{attribute 'qualified_only'}
{attribute 'strict'}
TYPE Command_State :
(
	Exekute := 0,
	Wate := 1,
	Complete := 2,
	Error := 3
) UINT;
END_TYPE

(* stored: Version 1.1.0.1, ProductVersion 3.1.4024.10
   DUT Command_State: Id {aac0a895-fc07-40b3-9211-4fea18b9fe15} *)
